FUNCTION_BLOCK PidController EXTENDS InstancePath IMPLEMENTS IController, IOut
VAR_INPUT
    parameters : PidParameters;
    cycleTime : Millisecond := 1;
END_VAR
VAR
    _error : LREAL;
    _previousError : LREAL;
    _deltaError : LREAL;
    _proportionalPart : LREAL;
    _integralPart : LREAL;
    _previousIntegralPart : LREAL;
    _differentialPart : LREAL;
    _differentialPartLimit : LREAL;
    _out : LREAL;
END_VAR

(* Limit the differential part. Convenient when the output is calculated for the first time.
The limit prevents it from having a very large value after the first call.*)
PROPERTY DifferentialPartLimit : LREAL
SET
_differentialPartLimit := DifferentialPartLimit;
END_SET
END_PROPERTY

PROPERTY Out : LREAL
GET
Out := _out;
END_GET
END_PROPERTY

(* Set previous integral part on first call. Prevents integrator term for needing to build up. *)
PROPERTY PreviousIntegralPart : LREAL
SET
_previousIntegralPart := PreviousIntegralPart;
END_SET
END_PROPERTY

METHOD Update : IOut
VAR_INPUT
    setpoint : LREAL;
    actual : LREAL;
END_VAR
_error := setpoint - actual;

_proportionalPart := parameters.Kp * _error;

_integralPart := _previousIntegralPart + parameters.Ki * _error * cycleTime;
_previousIntegralPart := _integralPart;

IF cycleTime <> 0 THEN
    _deltaError := (_error - _previousError) / cycleTime;
ELSE
    ADSLOGSTR(
        msgCtrlMask:=ADSLOG_MSGTYPE_ERROR,
        msgFmtStr:='%s: Enter a cycletime > 0!',
        strArg:=_path
    );
END_IF
IF _differentialPartLimit = 0 OR _deltaError <= _differentialPartLimit THEN
    _differentialPart := _deltaError * parameters.Kd;
END_IF
_previousError := _error;

_out := _proportionalPart + _integralPart + _differentialPart;
END_METHOD

END_FUNCTION_BLOCK

(* stored: Version 1.1.0.1, ProductVersion 3.1.4024.12
   POU PidController: Id {da73802b-2471-4be1-ae33-77c4e2eb36c6}, SpecialFunc None
   Property DifferentialPartLimit: Id {0e5fc49d-15ed-446b-b5c4-b8f8bc7054d6}
   Set Set: Id {ebaea50d-eb7b-45f8-9ebf-1ac59fe2b99d}
   Property Out: Id {15ef5403-f0db-4dd2-9900-07e6b4494afc}
   Get Get: Id {72cbacfe-7ca3-43fc-b241-9d203cf10514}
   Property PreviousIntegralPart: Id {84c7dc6b-7c17-4d37-ad09-62b2cacd0ffa}
   Set Set: Id {f9f66342-ded5-4cda-8f18-8e494b23a987}
   Method Update: Id {0846af4f-7650-4534-bc93-e3fdd529f31e} *)
